// TIA Portal V19 export
VAR_GLOBAL   // PLC tag table "U3Em0"
END_VAR
VAR_GLOBAL CONSTANT   // user constants
   U3EM0_JOB1 : DInt := 1;   // ID for Job
END_VAR
